FUNCTION_BLOCK FB_Verbinden EXTENDS FB_Basis
VAR_INPUT
	Reaktor			:I_Reaktor;
	Auswertung		:I_Auswertung;
END_VAR
VAR_OUTPUT
	
END_VAR
VAR
	
END_VAR

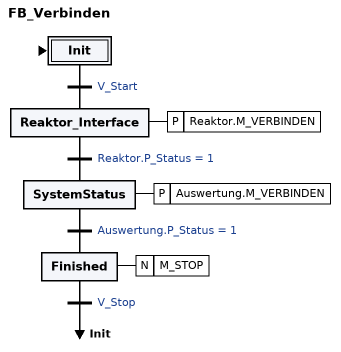
INITIAL_STEP Init:
END_STEP
TRANSITION FROM Init TO Reaktor_Interface
    := V_Start;
END_TRANSITION
STEP Reaktor_Interface:
    Reaktor.M_VERBINDEN(P);
END_STEP
TRANSITION FROM Reaktor_Interface TO SystemStatus_
    := Reaktor.P_Status = 1;
END_TRANSITION
STEP SystemStatus_:  // name as stored: SystemStatus 
    Auswertung.M_VERBINDEN(P);
END_STEP
TRANSITION FROM SystemStatus_ TO Finished
    := Auswertung.P_Status = 1;
END_TRANSITION
STEP Finished:
    M_STOP(N);
END_STEP
TRANSITION FROM Finished TO Init
    := V_Stop;
END_TRANSITION

END_FUNCTION_BLOCK

(* stored: Version 1.1.0.1, ProductVersion 3.1.4024.12
   POU FB_Verbinden: Id {88932e1c-43d3-46bb-93f4-7ca3981c47bc}, SpecialFunc None *)
